FUNCTION_BLOCK "LCB_12x_TablePositioning_V2"   // FB417, SCL
{ S7_Optimized_Access := 'FALSE' }
AUTHOR : Lenze
FAMILY : LCB
NAME : TabPosV2
VERSION : 2.0
   VAR_INPUT
      wHW_IO_Head : Hw_Io;
      i_stcAxisData : "stcLCB_12x_SetAxisData_Sw";
      xEnableInternalControl : Bool;
      iDriveType : Int;
      xDriveEnable : Bool;
      xDriveSetQsp : Bool;
      xResetError : Bool;
      xManualPos : Bool;
      xManualNeg : Bool;
      xHomingSet : Bool;
      xHomingStart : Bool;
      xHomingReset : Bool;
      xProfileStart : Bool;
      xProfileRestart : Bool;
      xProfileReset : Bool;
      xProfilePosStop : Bool;
      wProfileNumberSet : Word := W#16#1;
      xEnableSpeedOverride : Bool;
      rSpeedOverrideSet : Real := 1.0e+2;
      xEnablePositionTeach : Bool;
      rPositionSet : Real;
      xFreeCtrl_1 : Bool;
      xFreeCtrl_2 : Bool;
      xFreeCtrl_3 : Bool;
      xFreeCtrl_4 : Bool;
      xFreeCtrl_5 : Bool;
      xFreeCtrl_6 : Bool;
      xFreeCtrl_7 : Bool;
      xFreeCtrl_8 : Bool;
      wFreeCtrl_1 : Word;
   END_VAR
   VAR_OUTPUT
      xInternalControlActive : Bool;
      xError : Bool;
      xCommunicationOK : Bool;
      xDriveError : Bool;
      xDriveWarning : Bool;
      xDriveReady : Bool;
      xDriveEnabled : Bool;
      xDriveQspActive : Bool;
      xSpeedEqZero : Bool;
      xHomingActive : Bool;
      xHomingDone : Bool;
      xHomePosAvailable : Bool;
      xHomingSensorActivated : Bool;
      xManualActive : Bool;
      xProfileActive : Bool;
      xProfileDone : Bool;
      xProfileInTarget : Bool;
      xHW_LimitSwitchPos : Bool;
      xHW_LimitSwitchNeg : Bool;
      rSpeedActual : Real;
      rPosActual : Real;
      iReadError : Int;
      iWriteError : Int;
      xProfileIsStarting : Bool;   // Drive Application input xPosExecuteIsActive _xFreeState_1 ABS 7/2/2019
      xDirectionSpeedIsCcw : Bool;   // Drive is running anti-clockwise = reverse
      xDriveSafeTorqueOff : Bool;   // Drive Devicestate = SafeTorqueOff
      xFreeState_4 : Bool;
      xFreeState_5 : Bool;
      xFreeState_6 : Bool;
      xFreeState_7 : Bool;
      xFreeState_8 : Bool;
      wFreeState_1 : Word;
      xApplicationError : Bool;   // Table positioning application error, push reset
      xEnabledIsPositionTeach : Bool;   // bPosSetProfilePositionInside the drive
   END_VAR
   VAR
      wFirstPeripherieADR : Word;
      wProfileNumberSetIntern : Word;
      diActPos_p : DInt;
      rAccOverride : Real;
      xDriveEnable_IC : Bool;
      xDriveSetQsp_IC : Bool;
      xResetError_IC : Bool;
      xManualPos_IC : Bool;
      xManualNeg_IC : Bool;
      xHomingSet_IC : Bool;
      xHomingStart_IC : Bool;
      xHomingReset_IC : Bool;
      xProfileStart_IC : Bool;
      xProfileRestart_IC : Bool;
      xProfileReset_IC : Bool;
      xProfilePosStop_IC : Bool;
      xFreeCtrl_1_IC : Bool;
      xFreeCtrl_2_IC : Bool;
      xFreeCtrl_3_IC : Bool;
      xFreeCtrl_4_IC : Bool;
      xFreeCtrl_5_IC : Bool;
      xFreeCtrl_6_IC : Bool;
      xFreeCtrl_7_IC : Bool;
      xFreeCtrl_8_IC : Bool;
      wFreeCtrl_1_IC : Word;
      wProfileNumberSet_IC : Word := W#16#1;
      xwInput AT wProfileNumberSet_IC : Array[0..15] of Bool;
      xEnableSpeedOverride_IC : Bool;
      rSpeedOverrideSet_IC : Real := 1.0e+2;
      xEnablePositionTeach_IC : Bool;
      rPositionSet_IC : Real;
      wOUT : Word;
      xwOut AT wOUT : Array[0..15] of Bool;
      scInternalCtrl84 : Struct
         b8 : Bool;
         b9 : Bool;
         b10 : Bool;
         b11 : Bool;
         b12 : Bool;
         b13 : Bool;
         b14 : Bool;
         b15 : Bool;
         b0 : Bool;
         b1 : Bool;
         b2 : Bool;
         b3 : Bool;
         b4 : Bool;
         b5 : Bool;
         b6 : Bool;
         b7 : Bool;
         awInt : Array[2..6] of Word;
      END_STRUCT;
      scInternalState84 : Struct
         b8 : Bool;
         b9 : Bool;
         b10 : Bool;
         b11 : Bool;
         b12 : Bool;
         b13 : Bool;
         b14 : Bool;
         b15 : Bool;
         b0 : Bool;
         b1 : Bool;
         b2 : Bool;
         b3 : Bool;
         b4 : Bool;
         b5 : Bool;
         b6 : Bool;
         b7 : Bool;
         awInt : Array[2..6] of Word;
      END_STRUCT;
      scInternalCtrl94 : Struct
         b8 : Bool;
         b9 : Bool;
         b10 : Bool;
         b11 : Bool;
         b12 : Bool;
         b13 : Bool;
         b14 : Bool;
         b15 : Bool;
         b0 : Bool;
         b1 : Bool;
         b2 : Bool;
         b3 : Bool;
         b4 : Bool;
         b5 : Bool;
         b6 : Bool;
         b7 : Bool;
         awInt : Array[2..7] of Word;
      END_STRUCT;
      scInternalState94 : Struct
         b8 : Bool;
         b9 : Bool;
         b10 : Bool;
         b11 : Bool;
         b12 : Bool;
         b13 : Bool;
         b14 : Bool;
         b15 : Bool;
         b0 : Bool;
         b1 : Bool;
         b2 : Bool;
         b3 : Bool;
         b4 : Bool;
         b5 : Bool;
         b6 : Bool;
         b7 : Bool;
         awInt : Array[2..7] of Word;
      END_STRUCT;
      dwTemp : DWord;
      rTemp : Real;
      diSetPos : DInt;
   END_VAR
   VAR_TEMP
      Temp_1 : GEOADDR;
      RET : Int;
      tHW_IO : Hw_Any;
   END_VAR
BEGIN
   //#wFirstPeripherieADR:= INT_TO_WORD(#wHW_IO_Head);             
   #iReadError:=0;
   #iWriteError:=0;

   IF #xEnableInternalControl THEN                                    // Interne Steuerung des Reglers
       #xInternalControlActive:=True;
   ELSE                                                               // Steuerung des Reglers über Eingangsvariablen des Bausteins
       #xInternalControlActive:=False;
   END_IF;

   // Keine Interne Steuerung aktiv?
   IF NOT #xEnableInternalControl THEN
       // Eingangssignale auf interne Variablen kopieren
       #xDriveEnable_IC             := #xDriveEnable;
       #xDriveSetQsp_IC             := #xDriveSetQsp;
       #xResetError_IC              := #xResetError;
       #xManualPos_IC               := #xManualPos;
       #xManualNeg_IC               := #xManualNeg;
       #xHomingSet_IC               := #xHomingSet;
       #xHomingStart_IC             := #xHomingStart;
       #xHomingReset_IC             := #xHomingReset;
       #xProfileStart_IC            := #xProfileStart;
       #xProfileRestart_IC          := #xProfileRestart;
       #xProfileReset_IC            := #xProfileReset;
       #xProfilePosStop_IC          := #xProfilePosStop;
       #wProfileNumberSet_IC        := #wProfileNumberSet;
       #xEnableSpeedOverride_IC     := #xEnableSpeedOverride;
       #rSpeedOverrideSet_IC        := #rSpeedOverrideSet;
       #xEnablePositionTeach_IC     := #xEnablePositionTeach;
       #rPositionSet_IC             := #rPositionSet;
       #xFreeCtrl_1_IC              := #xFreeCtrl_1;
       #xFreeCtrl_2_IC              := #xFreeCtrl_2;
       #xFreeCtrl_3_IC              := #xFreeCtrl_3;
       #xFreeCtrl_4_IC              := #xFreeCtrl_4;
       #xFreeCtrl_5_IC              := #xFreeCtrl_5;
       #xFreeCtrl_6_IC              := #xFreeCtrl_6;
       #xFreeCtrl_7_IC              := #xFreeCtrl_7;
       #xFreeCtrl_8_IC              := #xFreeCtrl_8;
       #wFreeCtrl_1_IC              := #wFreeCtrl_1;
   END_IF;

   // HW-Kennung des IO-Moduls für 84/94 ermitteln

   #RET := LOG2GEO(LADDR := #wHW_IO_Head, GEOADDR := #Temp_1); // Aus HW-Kennung des Kopfmoduls den Steckplatz ermitteln
   #Temp_1.SLOT := #Temp_1.SLOT + 1;                           // Slotzähler erhöhen
   #RET := GEO2LOG(GEOADDR := #Temp_1, LADDR => #tHW_IO);      // Aus der Slotnummer die HW_Kennung des ersten Steckplatzes fü

   CASE #iDriveType OF

           // L-Force 8400 Highline / Topline / 8400 Protec Highline
           // Eingangsdaten vom Regler lesen
       2:
           #iReadError := DPRD_DAT(
                                   LADDR := #tHW_IO,
                                   RECORD => #scInternalState84);

           // Statusdaten zuweisen
           #xDriveError := #scInternalState84.b0;
           #xApplicationError := #scInternalState84.b1;
           #xEnabledIsPositionTeach := #scInternalState84.b2;
           #xDriveEnabled := NOT #scInternalState84.b3;
           #xDriveReady := #scInternalState84.b4;
           #xHomingSensorActivated := #scInternalState84.b5;
           #xHomingDone := #scInternalState84.b6;
           #xProfileDone := #scInternalState84.b7;
           #xProfileInTarget := #scInternalState84.b8;
           #xProfileActive := #scInternalState84.b9;
           #xHomePosAvailable := #scInternalState84.b10;
           #xSpeedEqZero := #scInternalState84.b11;
           #xHW_LimitSwitchNeg := #scInternalState84.b12;
           #xHW_LimitSwitchPos := #scInternalState84.b13;
           #xDriveQspActive := #scInternalState84.b14;
           #xDriveWarning := #scInternalState84.b15;

           #xHomingActive := #xHomingStart_IC AND #scInternalState84.b9;

           #rSpeedActual := LIMIT(MN := -199.99, IN := (INT_TO_REAL(WORD_TO_INT(#scInternalState84.awInt[5])) / 163.848), MX := 199.99);
           #diActPos_p := WORD_TO_DINT(#scInternalState84.awInt[3]) + DWORD_TO_DINT(SHL(IN := WORD_TO_DWORD(#scInternalState84.awInt[4]), N := 16));
           // ABS ;-)  #dwTemp := #AxisData.%DBD72;   // AxisData.rPosToUnits
           // ABS done :-) #rTemp := DWORD_TO_REAL(#dwTemp);
           #rPosActual := DINT_TO_REAL(#diActPos_p) * #i_stcAxisData.rPosToUnits;//#rTemp;

           #xProfileIsStarting := WORD_TO_INT((SHR(IN := #scInternalState84.awInt[2], N := 0) AND 16#0001)) > 0;
           #xDirectionSpeedIsCcw := WORD_TO_INT((SHR(IN := #scInternalState84.awInt[2], N := 1) AND 16#0001)) > 0;
           #xDriveSafeTorqueOff := #scInternalState84.awInt[6] >= 16#A00 AND #scInternalState84.awInt[6] <= 16#AFF; //Update TEF 20190917 Devicestate = SafeTorqueOff -> Binary xxxx 1010 xxxx xxxx
           #xFreeState_4 := WORD_TO_INT((SHR(IN := #scInternalState84.awInt[2], N := 3) AND 16#0001)) > 0;
           #xFreeState_5 := WORD_TO_INT((SHR(IN := #scInternalState84.awInt[2], N := 4) AND 16#0001)) > 0;
           #xFreeState_6 := WORD_TO_INT((SHR(IN := #scInternalState84.awInt[2], N := 5) AND 16#0001)) > 0;
           #xFreeState_7 := WORD_TO_INT((SHR(IN := #scInternalState84.awInt[2], N := 6) AND 16#0001)) > 0;
           #xFreeState_8 := WORD_TO_INT((SHR(IN := #scInternalState84.awInt[2], N := 7) AND 16#0001)) > 0;
           #wFreeState_1 := #scInternalState84.awInt[6];

           IF #xHomingStart_IC // Homing ?
               AND NOT #xProfileStart_IC
               AND NOT #xProfileRestart_IC
               AND NOT #xManualPos_IC
               AND NOT #xManualNeg_IC THEN
               // Auswahl 1. Profil für Referenzieren
               #wProfileNumberSet_IC := 1;
               #xManualActive := False;
           ELSIF ((#xManualPos_IC) OR (#xManualNeg_IC)) // Manual ?
               AND NOT #xProfileStart_IC
               AND NOT #xProfileRestart_IC
               AND NOT #xHomingStart_IC
               AND NOT #xHomingSet_IC THEN
               // Auswahl 0. Profil für Handfahren
               #wProfileNumberSet_IC := 0;
               #xManualActive := True;
           ELSE
               #xManualActive := False;

           END_IF;

           IF (NOT #xDriveEnable_IC) OR #xDriveError THEN
               // Merker für Positionieren zurücksetzen
               #xProfileStart_IC := FALSE;
               #xProfileRestart_IC := FALSE;
               #xProfileStart_IC := FALSE;
               #xProfileActive := FALSE;
               #xHomingStart_IC := False;
               #xHomingSet_IC := FALSE;
               #xManualPos_IC := FALSE;
               #xManualPos_IC := FALSE;
               // wProfileNumberSet_IC := 0;        Entfallen mit V1.1    
           END_IF;

           // Steuerdaten zuweisen
           #scInternalCtrl84.b0 := #xProfilePosStop_IC;
           #scInternalCtrl84.b1 := #xProfileRestart_IC AND NOT #xProfilePosStop_IC;
           #scInternalCtrl84.b2 := #xEnablePositionTeach_IC; //update ABS 6/2/2019 AND #xProfileStart_IC;
           #scInternalCtrl84.b3 := NOT #xDriveEnable_IC;
           #scInternalCtrl84.b4 := #xwInput[8];
           #scInternalCtrl84.b5 := #xwInput[9];
           #scInternalCtrl84.b6 := #xwInput[10];
           #scInternalCtrl84.b7 := #xwInput[11];
           #scInternalCtrl84.b8 := #xProfileStart_IC OR #xHomingStart_IC AND NOT #xProfilePosStop_IC;
           #scInternalCtrl84.b9 := #xEnableSpeedOverride_IC;
           #scInternalCtrl84.b10 := #xHomingSet_IC;
           #scInternalCtrl84.b11 := #xResetError_IC;
           #scInternalCtrl84.b12 := #xManualNeg_IC;
           #scInternalCtrl84.b13 := #xManualPos_IC;
           #scInternalCtrl84.b14 := #xHomingReset_IC;
           #scInternalCtrl84.b15 := #xDriveSetQsp_IC;

           // zuweisen der freien Controlbits
           #wOUT := 0;  // Initialisierung
           #xwOut[8] := #xFreeCtrl_1_IC;
           #xwOut[9] := #xFreeCtrl_2_IC;
           #xwOut[10] := #xFreeCtrl_3_IC;
           #xwOut[11] := #xFreeCtrl_4_IC;
           #xwOut[12] := #xFreeCtrl_5_IC;
           #xwOut[13] := #xFreeCtrl_6_IC;
           #xwOut[14] := #xFreeCtrl_7_IC;
           #xwOut[15] := #xFreeCtrl_8_IC;
           #scInternalCtrl84.awInt[2] := #wOUT;

           // limit rSpeedOverride
           #rSpeedOverrideSet_IC := LIMIT(MN := 0.0, IN := #rSpeedOverrideSet_IC, MX := 199.0);
           // scale and Write rSpeedOverride to drive
           IF #xEnableSpeedOverride_IC THEN
               #scInternalCtrl84.awInt[5] := INT_TO_WORD(REAL_TO_INT(#rSpeedOverrideSet_IC * 163.84));
           ELSE
               #scInternalCtrl84.awInt[5] := 16384;
           END_IF;
           //    convert units to increments    
          (* #dwTemp := 1; //#AxisData.%DBD68; // DB SetAxisData.rUnitsToPos
           #rTemp               :=DWORD_TO_REAL(#dwTemp);
          *)

           #diSetPos := REAL_TO_DINT(#rPositionSet_IC * #i_stcAxisData.rUnitsToPos);

           // write to drive*)
           #scInternalCtrl84.awInt[3] := DINT_TO_WORD(#diSetPos);
           #scInternalCtrl84.awInt[4] := DWORD_TO_WORD(SHR(IN := DINT_TO_DWORD(#diSetPos), N := 16));
           #scInternalCtrl84.awInt[6] := #wFreeCtrl_1_IC;

           // Ausgangsdaten zum Regler schreiben                         
           #iWriteError := DPWR_DAT(
                                    LADDR := #tHW_IO,
                                    RECORD := #scInternalCtrl84);

           #xError := (#iReadError <> 0) OR (#iWriteError <> 0)
           OR NOT ((#iDriveType <> 2) OR (#iDriveType <> 11))
           OR (WORD_TO_INT(#wProfileNumberSet_IC) > 15)
           OR (WORD_TO_INT(#wProfileNumberSet_IC) < 0);




           // L-Force 9400 Highline 
           // Eingangsdaten vom Regler lesen
       11:
           #iReadError := DPRD_DAT(
                                   LADDR := #tHW_IO,
                                   RECORD => #scInternalState94);

           // Statusdaten zuweisen
           #xDriveError := #scInternalState94.b0;
           #xDriveEnabled := NOT #scInternalState94.b1;
           #xDriveReady := #scInternalState94.b2;
           #xDriveQspActive := #scInternalState94.b3;
           #xSpeedEqZero := #scInternalState94.b4;
           #xHomingActive := #scInternalState94.b5;
           #xHomingDone := #scInternalState94.b6;
           #xHomePosAvailable := #scInternalState94.b7;
           #xManualActive := #scInternalState94.b8;
           #xDriveWarning := #scInternalState94.b9;
           #xProfileActive := #scInternalState94.b10;
           #xProfileDone := #scInternalState94.b11;
           #xProfileInTarget := #scInternalState94.b12;
           // xHomeSwitch      :=scInternalState94.b13;
           #xHW_LimitSwitchPos := #scInternalState94.b14;
           #xHW_LimitSwitchNeg := #scInternalState94.b15;

           #rSpeedActual := LIMIT(MN := -199.99, IN := (INT_TO_REAL(WORD_TO_INT(#scInternalState94.awInt[2])) / 163.848), MX := 199.99);
           #diActPos_p := WORD_TO_DINT(#scInternalState94.awInt[4]) + DWORD_TO_DINT(SHL(IN := WORD_TO_DWORD(#scInternalState94.awInt[3]), N := 16));
           // ABS;-) #dwTemp := #AxisData.%DBD72;   // AxisData.rPosToUnits
           // ABS :-) #rTemp := DWORD_TO_REAL(#dwTemp);
           #rPosActual := DINT_TO_REAL(#diActPos_p) * #i_stcAxisData.rPosToUnits;//#rTemp;

           #xProfileIsStarting := WORD_TO_INT((SHR(IN := #scInternalState94.awInt[6], N := 0) AND 16#0001)) > 0;
           #xDirectionSpeedIsCcw := WORD_TO_INT((SHR(IN := #scInternalState94.awInt[6], N := 1) AND 16#0001)) > 0;
           #xDriveSafeTorqueOff := WORD_TO_INT((SHR(IN := #scInternalState94.awInt[6], N := 2) AND 16#0001)) > 0;
           #xFreeState_4 := WORD_TO_INT((SHR(IN := #scInternalState94.awInt[6], N := 3) AND 16#0001)) > 0;
           #xFreeState_5 := WORD_TO_INT((SHR(IN := #scInternalState94.awInt[6], N := 4) AND 16#0001)) > 0;
           #xFreeState_6 := WORD_TO_INT((SHR(IN := #scInternalState94.awInt[6], N := 5) AND 16#0001)) > 0;
           #xFreeState_7 := WORD_TO_INT((SHR(IN := #scInternalState94.awInt[6], N := 6) AND 16#0001)) > 0;
           #xFreeState_8 := WORD_TO_INT((SHR(IN := #scInternalState94.awInt[6], N := 7) AND 16#0001)) > 0;
           #wFreeState_1 := #scInternalState94.awInt[5];

           IF (NOT #xDriveEnable_IC) OR #xDriveError THEN
               // Merker für Positionieren zurücksetzen
               #xProfileStart_IC := FALSE;
               #xProfileRestart_IC := FALSE;
               #xProfileStart_IC := FALSE;
               #xProfileActive := FALSE;
               #xHomingStart_IC := False;
               #xHomingSet_IC := FALSE;
               #xManualPos_IC := FALSE;
               #xManualPos_IC := FALSE;
               // wProfileNumberSet_IC := 1;    entfallen mit V1.1        
           END_IF;

           // Steuerdaten zuweisen
           #scInternalCtrl94.b0 := NOT #xDriveEnable_IC;
           #scInternalCtrl94.b1 := #xDriveSetQsp_IC;
           #scInternalCtrl94.b2 := #xEnablePositionTeach_IC;
           #scInternalCtrl94.b3 := #xHomingStart_IC;
           #scInternalCtrl94.b4 := #xHomingReset_IC;
           #scInternalCtrl94.b5 := #xProfileActive OR #xProfileStart_IC;
           #scInternalCtrl94.b6 := #xProfileStart_IC AND NOT #xProfilePosStop_IC;
           #scInternalCtrl94.b7 := #xProfileRestart_IC AND NOT #xProfilePosStop_IC;
           #scInternalCtrl94.b8 := #xProfileReset_IC;
           #scInternalCtrl94.b9 := #xEnableSpeedOverride_IC;
           #scInternalCtrl94.b10 := #xResetError_IC;
           #scInternalCtrl94.b11 := False; // Spare Set Error
           #scInternalCtrl94.b12 := #xHomingSet_IC;
           #scInternalCtrl94.b13 := False; // Spare
           #scInternalCtrl94.b14 := #xManualPos_IC;
           #scInternalCtrl94.b15 := #xManualNeg_IC;

           // zuweisen der freien Controlbits
           #wOUT := 0;  // Initialisierung
           #xwOut[8] := #xFreeCtrl_1_IC;
           #xwOut[9] := #xFreeCtrl_2_IC;
           #xwOut[10] := #xFreeCtrl_3_IC;
           #xwOut[11] := #xFreeCtrl_4_IC;
           #xwOut[12] := #xFreeCtrl_5_IC;
           #xwOut[13] := #xFreeCtrl_6_IC;
           #xwOut[14] := #xFreeCtrl_7_IC;
           #xwOut[15] := #xFreeCtrl_8_IC;
           #scInternalCtrl94.awInt[6] := #wOUT;
           #scInternalCtrl94.awInt[7] := #wFreeCtrl_1_IC;

           // limit rSpeedOverride
           #rSpeedOverrideSet_IC := LIMIT(MN := 0.0, IN := #rSpeedOverrideSet_IC, MX := 199.0);
           // scale and Write rSpeedOverride to drive
           IF #xEnableSpeedOverride_IC THEN
               #scInternalCtrl94.awInt[2] := INT_TO_WORD(REAL_TO_INT(#rSpeedOverrideSet_IC * 163.84));
           ELSE
               #scInternalCtrl94.awInt[2] := 16384;
           END_IF;
           // convert units to increments    
           //ABS :-)  #dwTemp := #AxisData.%DBD68; // DB SetAxisData.rUnitsToPos
           //ABS :-)  #rTemp := DWORD_TO_REAL(#dwTemp);
           #diSetPos := REAL_TO_DINT(#rPositionSet_IC * #i_stcAxisData.rUnitsToPos);//#rTemp);

           // write to drive*)
           #scInternalCtrl94.awInt[4] := DINT_TO_WORD(#diSetPos);
           #scInternalCtrl94.awInt[3] := DWORD_TO_WORD(SHR(IN := DINT_TO_DWORD(#diSetPos), N := 16));

           // limit  ProfileNumber and write To Drive      
           #scInternalCtrl94.awInt[5] := INT_TO_WORD(LIMIT(MN := 1, IN := WORD_TO_INT(#wProfileNumberSet_IC), MX := 75));

           // Ausgangsdaten zum Regler schreiben                         
           #iWriteError := DPWR_DAT(
                                    LADDR := #tHW_IO,
                                    RECORD := #scInternalCtrl94);

           #xError := (#iReadError <> 0) OR (#iWriteError <> 0)
           OR NOT ((#iDriveType <> 1) OR (#iDriveType <> 2) OR (#iDriveType <> 11))
           OR (WORD_TO_INT(#wProfileNumberSet_IC) > 75)
           OR (WORD_TO_INT(#wProfileNumberSet_IC) < 1);

       ELSE:
           #xError := True;
   END_CASE;

   IF (#iReadError <> 0) OR (#iWriteError <> 0) THEN
       #xCommunicationOK:=false;
   ELSE
       #xCommunicationOK:=True;
   END_IF;
END_FUNCTION_BLOCK

FUNCTION_BLOCK "LCB_12x_SetAxisData"   // FB443, SCL
{ S7_Optimized_Access := 'FALSE' }
AUTHOR : Lenze
FAMILY : LCB
NAME : SetAxisD
VERSION : 1.0
   VAR_INPUT
      rFeedConstant : Real := 3.6e+2;
      rCycleLength : Real := 3.6e+2;
      diGearNumerator : DInt := L#1;
      diGearDenominator : DInt := L#1;
      rReferenceSpeed : Real := 1.8e+5;
      rReferenceTorque : Real := 1.0e+0;
      sAxisName : String[16] := 'MyAxis';
      rResolution : Real := 16.0;
   END_VAR
   VAR_OUTPUT
      AxisData : "stcLCB_12x_SetAxisData_Sw";
   END_VAR
   VAR_IN_OUT
      xModeUnlimited : Bool := TRUE;
      xModeLimited : Bool;
      xModeModulo : Bool;
   END_VAR
   VAR
      rInvFeedConstant : Real;
      diReferenceSpeed_s : DInt;
      rEncoderGear : Real;
      rInvEncoderGear : Real;
      diCycleLength_p : DInt;
      rUnitsToPos : Real;
      rPosToUnits : Real;
      rUnitsToSpeed : Real;
      rSpeedToUnits : Real;
      rTimeUnit : Real := 6.0e+1;
      rFeedConstantOld : Real;
      rCycleLengthOld : Real;
      diGearNumeratorOld : DInt := L#2;
      diGearDenominatorOld : DInt := L#2;
      rReferenceSpeedOld : Real;
      rResolutionOld : Real := 1.0;
      xModeUnlimitedOld : Bool;
      xModeLimitedOld : Bool;
      xModeModuloOld : Bool;
   END_VAR
BEGIN

       IF #xModeUnlimited= True THEN #xModeLimited:= False; #xModeModulo:= False;
           ELSIF #xModeLimited= True THEN #xModeUnlimited:= False; #xModeModulo:= False;
               ELSIF #xModeModulo= True THEN #xModeUnlimited:= False; #xModeLimited:= False;
       END_IF; 
       IF ((#rFeedConstantOld <> #rFeedConstant) OR
           (#diGearNumeratorOld <> #diGearNumerator) OR
           (#diGearDenominatorOld <> #diGearDenominator) OR
           (#rCycleLengthOld <> #rCycleLength) OR
           (#xModeUnlimitedOld <> #xModeUnlimited) OR
           (#xModeLimitedOld <> #xModeLimited) OR
           (#xModeModuloOld <> #xModeModulo) OR
           (#rResolutionOld <> #rResolution) OR
           (#rReferenceSpeedOld <> #rReferenceSpeed)) THEN


           #rInvFeedConstant := 1.0 / #rFeedConstant;

       (* Achsdatenberechnung starten *)
       (* Getriebefaktor *)
           #rEncoderGear:=DINT_TO_REAL(#diGearNumerator) / DINT_TO_REAL(#diGearDenominator);
           #rInvEncoderGear:= 1.0 / #rEncoderGear;
       (* Umrechenfaktor Units -> _p bestimmen *)
           #rUnitsToPos := (#rInvFeedConstant * #rEncoderGear) * (2**#rResolution);
       (* Umrechenfaktor _p -> Units bestimmen *)
           #rPosToUnits := 1.0 / #rUnitsToPos;
       (* Umrechenfaktor Units->_s bestimmen *)
           #rUnitsToSpeed := #rInvFeedConstant * #rEncoderGear;
     //  (* mal 2^32 (eine Umdrehung) *)
     //      rUnitsToSpeed := rUnitsToSpeed * 2**32;
       (* durch Zeiteinheit teilen *)
           #rUnitsToSpeed := #rUnitsToSpeed * #rTimeUnit;
       (* Umrechenfaktor _s -> Units bestimmen *)
           #rSpeedToUnits := 1.0 / #rUnitsToSpeed;
       (*Referenzgeschwindigkeit bestimmen *)
           #diReferenceSpeed_s := REAL_TO_DINT(#rReferenceSpeed * #rUnitsToSpeed);

           IF #xModeModulo THEN
               #diCycleLength_p := REAL_TO_DINT(#rCycleLength * #rUnitsToPos) ;
           ELSE
               #diCycleLength_p := 0;
           END_IF;

       // sichern der aktuellen Werte für Änderungsvergleich
           #rFeedConstantOld     :=#rFeedConstant     ;
           #rCycleLengthOld      :=#rCycleLength      ;    
           #diGearNumeratorOld   :=#diGearNumerator   ;
           #diGearDenominatorOld :=#diGearDenominator ;
           #rReferenceSpeedOld   :=#rReferenceSpeed   ;
           #xModeUnlimitedOld    :=#xModeUnlimited    ;
           #xModeLimitedOld      :=#xModeLimited      ;
           #xModeModuloOld       :=#xModeModulo       ;
           #rResolutionOld      :=#rResolution      ;  

       END_IF;

   //Write to global output status
       #AxisData.rUnitsToPos := #rUnitsToPos;
       #AxisData.rPosToUnits := #rPosToUnits;
END_FUNCTION_BLOCK

(* ===== HMI "HMI_RT_1" =====
system functions are stored by id; their names below are inferred from use
connection "HMI_Connection_1": ETHERNET, S7_1200_OMS

HMI tags "Default tag table"
   "VIS_CmDrvSerPos_stc_Indicators_Status_IsEnabled" : Bool = PLC VIS_CmDrvSerPos.stc.Indicators.Status.IsEnabled, 1 s
   "VIS_CmDrvSerPos_stc_Commands_Enable" : Bool = PLC VIS_CmDrvSerPos.stc.Commands.Enable, 1 s
   "VIS_CmDrvSerPos_stc_Commands_JogFwdCwUpLoading" : Bool = PLC VIS_CmDrvSerPos.stc.Commands.JogFwdCwUpLoading, 1 s
   "VIS_CmDrvSerPos_stc_Commands_JogRevCcwDownUnloading" : Bool = PLC VIS_CmDrvSerPos.stc.Commands.JogRevCcwDownUnloading, 1 s
   "VIS_CmDrvSerPos_stc_Indicators_Status_BusyJogFwdCwUpLoading" : Bool = PLC VIS_CmDrvSerPos.stc.Indicators.Status.BusyJogFwdCwUpLoading, 1 s
   "VIS_CmDrvSerPos_stc_Indicators_Status_BusyJogRevCcwDownUnloading" : Bool = PLC VIS_CmDrvSerPos.stc.Indicators.Status.BusyJogRevCcwDownUnloading, 1 s
   "VIS_CmDrvSerPos_stc_Commands_PbReset" : Bool = PLC VIS_CmDrvSerPos.stc.Commands.PbReset, 1 s
   "VIS_CmDrvSerPos_stc_Indicators_PushButtons_PbReset" : Bool = PLC VIS_CmDrvSerPos.stc.Indicators.PushButtons.PbReset, 1 s
   "VIS_CmDrvSerPos_stc_Commands_StartHoming" : Bool = PLC VIS_CmDrvSerPos.stc.Commands.StartHoming, 1 s
   "VIS_CmDrvSerPos_stc_Indicators_Status_IsHomed" : Bool = PLC VIS_CmDrvSerPos.stc.Indicators.Status.IsHomed, 1 s
   "VIS_CmDrvSerPos_stc_Commands_StartExecuteAutomatic" : Bool = PLC VIS_CmDrvSerPos.stc.Commands.StartExecuteAutomatic, 1 s
   "VIS_CmDrvSerPos_stc_Commands_StopHoming" : Bool = PLC VIS_CmDrvSerPos.stc.Commands.StopHoming, 1 s
   "VIS_CmDrvSerPos_stc_Recipe_rSpPosition_Units" : Real = PLC VIS_CmDrvSerPos.stc.Recipe.rSpPosition_Units, 1 s
   "VIS_CmDrvSerPos_stc_SD_ProcessValue_rPvPosition_Units" : Real = PLC VIS_CmDrvSerPos.stc.SD.ProcessValue.rPvPosition_Units, 1 s
   "VIS_CmDrvSerPos_stc_Indicators_PushButtons_StopHoming" : Bool = PLC VIS_CmDrvSerPos.stc.Indicators.PushButtons.StopHoming, 1 s
   "VIS_CmDrvSerPos_stc_Indicators_PushButtons_StartHoming" : Bool = PLC VIS_CmDrvSerPos.stc.Indicators.PushButtons.StartHoming, 1 s
   "VIS_CmDrvSerPos_stc_Indicators_PushButtons_StartExecuteAutomatic" : Bool = PLC VIS_CmDrvSerPos.stc.Indicators.PushButtons.StartExecuteAutomatic, 1 s
   "VIS_CmDrvSerPos_stc_Indicators_Status_IsAtTargetPosSpeed" : Bool = PLC VIS_CmDrvSerPos.stc.Indicators.Status.IsAtTargetPosSpeed, 1 s
   "VIS_CmDrvSerPos_stc_Commands_StopExecuteAutomatic" : Bool = PLC VIS_CmDrvSerPos.stc.Commands.StopExecuteAutomatic, 1 s
   "VIS_CmDrvSerPos_stc_Indicators_PushButtons_StopExecuteAutomatic" : Bool = PLC VIS_CmDrvSerPos.stc.Indicators.PushButtons.StopExecuteAutomatic, 1 s
   "VIS_CmDrvSerPos_stc_SD_ErrorWarning_bErrorTripped" : Bool = PLC VIS_CmDrvSerPos.stc.SD.ErrorWarning.bErrorTripped, 1 s
   "VIS_CmDrvSerPos_stc_SD_ErrorWarning_bWarningTripped" : Bool = PLC VIS_CmDrvSerPos.stc.SD.ErrorWarning.bWarningTripped, 1 s
   "VIS_CmDrvSerPos_stc_SD_bRFR" : Bool = PLC VIS_CmDrvSerPos.stc.SD.bRFR, 1 s
   "VIS_CmDrvSerPos_stc_SD_ErrorWarning_wError" : Word = PLC VIS_CmDrvSerPos.stc.SD.ErrorWarning.wError, 1 s
   "VIS_CmDrvSerPos_stc_SD_ErrorWarning_wWarning" : Word = PLC VIS_CmDrvSerPos.stc.SD.ErrorWarning.wWarning, 1 s
   "VIS_CmDrvSerPos_stc_bLimitsSwitchPositiveActivated" : Bool = PLC VIS_CmDrvSerPos.stc.bLimitsSwitchPositiveActivated, 1 s
   "VIS_CmDrvSerPos_stc_bLimitsSwitchNegativeActivated" : Bool = PLC VIS_CmDrvSerPos.stc.bLimitsSwitchNegativeActivated, 1 s
   "VIS_CmDrvSerPos_stc_bHomingSensorActivated" : Bool = PLC VIS_CmDrvSerPos.stc.bHomingSensorActivated, 1 s
   "VIS_CmDrvSerPos_stc_CD_iModeSet" : Int = PLC VIS_CmDrvSerPos.stc.CD.iModeSet, 1 s
   "VIS_CmDrvSerPos_stc_Commands_ModeChange" : Bool = PLC VIS_CmDrvSerPos.stc.Commands.ModeChange, 1 s
   "DB_CmDrvSerPos_CD_iModeSet" : Int = PLC DB_CmDrvSerPos.CD.iModeSet, 1 s
   "DB_CmDrvSerPos_CD_Commands_ModeChange" : Bool = PLC DB_CmDrvSerPos.CD.Commands.ModeChange, 1 s
   "VIS_CmDrvSerPos_stc_SD_iModeActual" : Int = PLC VIS_CmDrvSerPos.stc.SD.iModeActual, 1 s
   "VIS_CmDrvSerPos_stc_Commands_Disable" : Bool = PLC VIS_CmDrvSerPos.stc.Commands.Disable, 1 s
   "VIS_CmDrvSerPos_stc_SD_iModuleState" : Int = PLC VIS_CmDrvSerPos.stc.SD.iModuleState, 1 s
   "VIS_CmDrvSerPos_stc_SD_bExecuting" : Bool = PLC VIS_CmDrvSerPos.stc.SD.bExecuting, 1 s
   "VIS_CmDrvSerPos_stc_Commands_EnableReleaseErrorWarning" : Bool = PLC VIS_CmDrvSerPos.stc.Commands.EnableReleaseErrorWarning, 1 s
   "VIS_CmDrvSerPos_stc_Commands_DisableReleaseErrorWarning" : Bool = PLC VIS_CmDrvSerPos.stc.Commands.DisableReleaseErrorWarning, 1 s
   "VIS_CmDrvSerPos_stc_Commands_ExecuteLoadRecipe" : Bool = PLC VIS_CmDrvSerPos.stc.Commands.ExecuteLoadRecipe, 1 s
   "VIS_CmDrvSerPos_stc_SD_ErrorWarningReleased" : Bool = PLC VIS_CmDrvSerPos.stc.SD.ErrorWarningReleased AT %DB1.DBX0.0, 1 s
   "di_FeedbackEmStop" : Bool = PLC di_FeedbackEmStop AT %I0.4, 1 s
   "VIS_CmDrvSerPos_stc_Indicators_PushButtons_Enable" : Bool = PLC VIS_CmDrvSerPos.stc.Indicators.PushButtons.Enable, 1 s
   "VIS_CmDrvSerPos_stc_Indicators_PushButtons_Disable" : Bool = PLC VIS_CmDrvSerPos.stc.Indicators.PushButtons.Disable, 1 s
   "VIS_CmDrvSerPos_stc_Indicators_PushButtons_ExecuteLoadRecipe" : Bool = PLC VIS_CmDrvSerPos.stc.Indicators.PushButtons.ExecuteLoadRecipe, 1 s
   "VIS_CmDrvSerPos_stc_Settings_rSpLimitH_Units" : Real = PLC VIS_CmDrvSerPos.stc.Settings.rSpLimitH_Units, 1 s
   "VIS_CmDrvSerPos_stc_Settings_rSpLimitL_Units" : Real = PLC VIS_CmDrvSerPos.stc.Settings.rSpLimitL_Units, 1 s
   "VIS_CmDrvSerPos_stc_Settings_rSpPositionOffset_Units" : Real = PLC VIS_CmDrvSerPos.stc.Settings.rSpPositionOffset_Units, 1 s
   "VIS_CmDrvSerPos_stc_Settings_iSetUnits" : Int = PLC VIS_CmDrvSerPos.stc.Settings.iSetUnits, 1 s

text list "Mode": 0 'Undefined'; 1 'AutoInline'; 2 'AutoStandalone'; 3 'Manual'; 4 'Service'; 5 'SingleStep'

screen "Screen_1" 800x480, template "Template_1"
   Rectangle "Rectangle_1" at 17,147 size 20x90
      Appearance <- "VIS_CmDrvSerPos_stc_Indicators_PushButtons_Enable"
   Button "Button_1" at 34,147 size 150x90; TextOff 'Enable'
      on Release: ResetBit("VIS_CmDrvSerPos_stc_Commands_Enable")
      on Press: SetBit("VIS_CmDrvSerPos_stc_Commands_Enable")
   Rectangle "Rectangle_2" at 196,376 size 20x90
      Appearance <- "VIS_CmDrvSerPos_stc_Indicators_Status_BusyJogFwdCwUpLoading"
   Button "Button_2" at 213,376 size 150x90; TextOff 'Fwd/Up'
      on Release: ResetBit("VIS_CmDrvSerPos_stc_Commands_JogFwdCwUpLoading")
      on Press: SetBit("VIS_CmDrvSerPos_stc_Commands_JogFwdCwUpLoading")
   Rectangle "Rectangle_3" at 14,376 size 20x90
      Appearance <- "VIS_CmDrvSerPos_stc_Indicators_Status_BusyJogRevCcwDownUnloading"
   Button "Button_3" at 31,376 size 150x90; TextOff 'Rev/Down'
      on Release: ResetBit("VIS_CmDrvSerPos_stc_Commands_JogRevCcwDownUnloading")
      on Press: SetBit("VIS_CmDrvSerPos_stc_Commands_JogRevCcwDownUnloading")
   Rectangle "Rectangle_4" at 17,246 size 20x90
      Appearance <- "VIS_CmDrvSerPos_stc_Indicators_PushButtons_PbReset"
   Button "Button_4" at 34,246 size 150x90; TextOff 'Reset'
      on Release: ResetBit("VIS_CmDrvSerPos_stc_Commands_PbReset")
      on Press: SetBit("VIS_CmDrvSerPos_stc_Commands_PbReset")
   Button "Button_5" at 213,246 size 150x90; TextOff 'QuickStop'
   Rectangle "Rectangle_6" at 389,376 size 20x90
      Appearance <- "VIS_CmDrvSerPos_stc_Indicators_PushButtons_StartHoming"
   Button "Button_6" at 406,376 size 150x90; TextOff 'Start'
      on Release: ResetBit("VIS_CmDrvSerPos_stc_Commands_StartHoming")
      on Press: SetBit("VIS_CmDrvSerPos_stc_Commands_StartHoming")
   Rectangle "Rectangle_7" at 390,150 size 20x90
      Appearance <- "VIS_CmDrvSerPos_stc_Indicators_PushButtons_StartExecuteAutomatic"
   Button "Button_7" at 407,150 size 150x90; TextOff 'Enable'
      on Release: ResetBit("VIS_CmDrvSerPos_stc_Commands_StartExecuteAutomatic")
      on Press: SetBit("VIS_CmDrvSerPos_stc_Commands_StartExecuteAutomatic")
   TextField "Text field_1" at 525,349 size 73x23; Text 'Homing'
   TextField "Text field_2" at 169,349 size 36x23; Text 'Jog'
   Button "Button_8" at 569,376 size 150x90; TextOff 'Stop'
      on Release: ResetBit("VIS_CmDrvSerPos_stc_Commands_StopHoming")
      on Press: SetBit("VIS_CmDrvSerPos_stc_Commands_StopHoming")
   TextField "Text field_3" at 471,121 size 152x23; Text 'Position Control'
   IOField "I/O field_1" at 414,248 size 141x39; FormatPattern s999.9; Unit mm
      ProcessValue <- "VIS_CmDrvSerPos_stc_Recipe_rSpPosition_Units"
   IOField "I/O field_2" at 415,293 size 140x41; FormatPattern s999.9; Unit mm
      ProcessValue <- "VIS_CmDrvSerPos_stc_SD_ProcessValue_rPvPosition_Units"
   Rectangle "Rectangle_12" at 620,350 size 20x24
      Appearance <- "VIS_CmDrvSerPos_stc_Indicators_Status_IsHomed"
   Button "Button_9" at 573,150 size 150x90; TextOff 'Disable'
      on Release: ResetBit("VIS_CmDrvSerPos_stc_Commands_StopExecuteAutomatic")
      on Press: SetBit("VIS_CmDrvSerPos_stc_Commands_StopExecuteAutomatic")
   Rectangle "Rectangle_14" at 716,150 size 20x90
      Appearance <- "VIS_CmDrvSerPos_stc_Indicators_PushButtons_StopExecuteAutomatic"
   TextField "Text field_6" at 385,255 size 28x23; Text 'SP'
   TextField "Text field_7" at 385,300 size 29x23; Text 'PV'
   Button "Button_10" at 6,52 size 739x52; TextOff 'Enable'
   TextField "Text field_8" at 315,17 size 143x23; Text 'CmDriveSerPos'
   TextField "Text field_9" at 151,119 size 76x23; Text 'General'
   Rectangle "Rectangle_10" at 716,376 size 20x90
      Appearance <- "VIS_CmDrvSerPos_stc_Indicators_PushButtons_StopHoming"
   Button "Button_11" at 747,417 size 51x56; TextOff 'Enable'; PictureOff "Down_Arrow"
      on Release: ActivateScreen("Screen_2", 0)
   Button "Button_12" at 747,112 size 51x56; TextOff 'Enable'; PictureOff "Up_Arrow"
      on Release: ActivateScreen("Screen_2", 0)
   TextField "Text field_10" at 772,280 size 16x23; Text '3'
   TextField "Text field_11" at 751,280 size 16x23; Text '1'
   Button "Button_13" at 747,52 size 50x52; TextOff 'CmValveCtrl'; PictureOff "Home"
      on Release: ActivateScreen("Main_Screen", 0)
   IOField "I/O field_3" at 18,117 size 44x26; FormatPattern 9999
      ProcessValue <- "VIS_CmDrvSerPos_stc_SD_iModuleState"
   Button "Button_15" at 573,246 size 145x40; TextOff 'Single Step'
      on Release: ResetBit("VIS_CmDrvSerPos_stc_Commands_ExecuteLoadRecipe")
      on Press: SetBit("VIS_CmDrvSerPos_stc_Commands_ExecuteLoadRecipe")
   TextField "Text field_4" at 645,352 size 94x18; Text 'HomingDone'
   Rectangle "Rectangle_16" at 620,122 size 20x24
      Appearance <- "VIS_CmDrvSerPos_stc_Indicators_Status_IsAtTargetPosSpeed"
   TextField "Text field_5" at 645,125 size 66x18; Text 'InTarget'
   Rectangle "Rectangle_13" at 254,119 size 20x24
      Appearance <- "VIS_CmDrvSerPos_stc_Indicators_Status_IsEnabled"
   TextField "Text field_12" at 279,122 size 60x18; Text 'Enabled'
   Rectangle "Rectangle_17" at 196,147 size 20x90
      Appearance <- "VIS_CmDrvSerPos_stc_Indicators_PushButtons_Disable"
   Button "Button_14" at 212,147 size 150x90; TextOff 'Disable'
      on Release: ResetBit("VIS_CmDrvSerPos_stc_Commands_Disable")
      on Press: SetBit("VIS_CmDrvSerPos_stc_Commands_Disable")
   Rectangle "Rectangle_18" at 716,246 size 20x90
      Appearance <- "VIS_CmDrvSerPos_stc_Indicators_PushButtons_ExecuteLoadRecipe"
   Button "Button_16" at 573,296 size 145x40; TextOff 'Automatic'
      on Press: SetBit("VIS_CmDrvSerPos_stc_Commands_ExecuteLoadRecipe")

screen "Screen_2" 800x480, template "Template_1"
   TextField "Text field_3" at 458,119 size 232x23; Text 'Status Sequence Stepper'
   Button "Button_10" at 6,52 size 739x52; TextOff 'Enable'
   TextField "Text field_8" at 315,17 size 143x23; Text 'CmDriveSerPos'
   TextField "Text field_9" at 149,119 size 108x23; Text 'Status OEM'
   Button "Button_12" at 747,417 size 51x56; TextOff 'Enable'; PictureOff "Down_Arrow"
      on Release: ActivateScreen("Screen_3", 0)
   Button "Button_13" at 747,112 size 51x56; TextOff 'Enable'; PictureOff "Up_Arrow"
      on Release: ActivateScreen("Screen_1", 0)
   TextField "Text field_10" at 772,280 size 16x23; Text '3'
   TextField "Text field_11" at 750,280 size 16x23; Text '2'
   Ellipse "Ellipse_1" at 397,149 size 28x28
      Appearance <- "VIS_CmDrvSerPos_stc_Indicators_Status_IsEnabled"
   TextField "Text field_2" at 435,152 size 77x23; Text 'Enabled'
   Ellipse "Ellipse_2" at 24,184 size 28x28
      Appearance <- "VIS_CmDrvSerPos_stc_SD_ErrorWarning_bErrorTripped"
   TextField "Text field_12" at 60,187 size 51x23; Text 'Error'
   Ellipse "Ellipse_3" at 398,189 size 28x28
      Appearance <- "VIS_CmDrvSerPos_stc_Indicators_Status_BusyJogRevCcwDownUnloading"
   TextField "Text field_13" at 436,190 size 125x23; Text 'Jog Fwd busy'
   Ellipse "Ellipse_4" at 397,229 size 28x28
      Appearance <- "VIS_CmDrvSerPos_stc_Indicators_Status_BusyJogRevCcwDownUnloading"
   TextField "Text field_14" at 437,229 size 123x23; Text 'Jog Rev busy'
   Ellipse "Ellipse_5" at 397,267 size 28x28
      Appearance <- "VIS_CmDrvSerPos_stc_SD_iModuleState"
   TextField "Text field_1" at 440,267 size 120x23; Text 'Homing busy'
   Ellipse "Ellipse_6" at 397,303 size 28x28
      Appearance <- "VIS_CmDrvSerPos_stc_SD_iModuleState"
   TextField "Text field_4" at 441,306 size 166x23; Text 'Position Ctrl busy'
   Ellipse "Ellipse_7" at 24,146 size 28x28
      Appearance <- "VIS_CmDrvSerPos_stc_SD_ErrorWarning_bWarningTripped"
   TextField "Text field_5" at 59,149 size 80x23; Text 'Warning'
   Ellipse "Ellipse_8" at 23,261 size 28x28
      Appearance <- "VIS_CmDrvSerPos_stc_SD_bRFR"
   TextField "Text field_6" at 60,264 size 115x23; Text 'Drive Ready'
   Ellipse "Ellipse_9" at 23,222 size 28x28
      Appearance <- "VIS_CmDrvSerPos_stc_Indicators_Status_IsEnabled"
   TextField "Text field_7" at 60,225 size 131x23; Text 'Drive Enabled'
   Ellipse "Ellipse_10" at 23,302 size 28x28
      Appearance <- "VIS_CmDrvSerPos_stc_Indicators_Status_IsHomed"
   TextField "Text field_15" at 61,306 size 67x23; Text 'Homed'
   IOField "I/O field_1" at 162,378 size 80x40; FormatPattern 99999
      ProcessValue <- "VIS_CmDrvSerPos_stc_SD_ErrorWarning_wWarning"
   TextField "Text field_17" at 18,388 size 135x23; Text 'Warning code:'
   IOField "I/O field_2" at 162,425 size 80x40; FormatPattern 99999
      ProcessValue <- "VIS_CmDrvSerPos_stc_SD_ErrorWarning_wError"
   TextField "Text field_16" at 20,431 size 106x23; Text 'Error code:'
   Ellipse "Ellipse_11" at 397,359 size 28x28
      Appearance <- "VIS_CmDrvSerPos_stc_bLimitsSwitchPositiveActivated"
   TextField "Text field_18" at 441,362 size 155x23; Text 'Limit Switch Pos'
   Ellipse "Ellipse_12" at 397,394 size 28x28
      Appearance <- "VIS_CmDrvSerPos_stc_bLimitsSwitchNegativeActivated"
   TextField "Text field_19" at 441,397 size 158x23; Text 'Limit Switch Neg'
   Ellipse "Ellipse_13" at 397,429 size 28x28
      Appearance <- "VIS_CmDrvSerPos_stc_bHomingSensorActivated"
   TextField "Text field_20" at 442,432 size 140x23; Text 'Homing Sensor'
   Button "Button_1" at 747,52 size 50x52; TextOff 'CmValveCtrl'; PictureOff "Home"
      on Release: ActivateScreen("Main_Screen", 0)
   Ellipse "Ellipse_14" at 22,341 size 28x28
      Appearance <- "VIS_CmDrvSerPos_stc_SD_bExecuting"
   TextField "Text field_21" at 60,345 size 94x23; Text 'Executing'
   Button "Button_2" at 176,155 size 81x57; TextOff 'Enable'
      on Release: ResetBit("VIS_CmDrvSerPos_stc_Commands_EnableReleaseErrorWarning")
      on Press: SetBit("VIS_CmDrvSerPos_stc_Commands_EnableReleaseErrorWarning")
   Button "Button_3" at 268,155 size 81x57; TextOff 'Disable'
      on Release: ResetBit("VIS_CmDrvSerPos_stc_Commands_DisableReleaseErrorWarning")
      on Press: SetBit("VIS_CmDrvSerPos_stc_Commands_DisableReleaseErrorWarning")
   Rectangle "Rectangle_13" at 160,154 size 20x58
      Appearance <- "VIS_CmDrvSerPos_stc_SD_ErrorWarningReleased"

Template "Template_1" 800x480
   TextField "Text field_1" at 762,279 size 15x23; Text '/'

screen "HMI_Settings" 800x480
   TextField "Text field_8" at 346,17 size 122x23; Text 'HMI Settings'
   Button "HmiScreenItemData" at 23,131 size 159x47; TextOn 'SIMATIC PLC system diagnos...'; TextOff 'SIMATIC PLC system diagnos...'; PictureOn "Navigates to SIMATIC PLC system diagnostics for TP700 Comfort 15.1.0.0"; PictureOff "Navigates to SIMATIC PLC system diagnostics for TP700 Comfort 15.1.0.0"
   Button "HmiScreenItemData_1" at 23,190 size 159x47; TextOn 'Project information'; TextOff 'Project information'; PictureOn "Navigates to Project information for TP700 Comfort 15.1.0.0"; PictureOff "Navigates to Project information for TP700 Comfort 15.1.0.0"
   Button "HmiScreenItemData_2" at 23,249 size 159x47; TextOn 'System settings'; TextOff 'System settings'; PictureOn "Navigates to System settings for TP700 Comfort 15.1.0.0"; PictureOff "Navigates to System settings for TP700 Comfort 15.1.0.0"
   Button "HmiScreenItemData_3" at 23,308 size 159x47; TextOn 'User administration'; TextOff 'User administration'; PictureOn "Navigates to User administration for TP700 Comfort 15.1.0.0"; PictureOff "Navigates to User administration for TP700 Comfort 15.1.0.0"
      on Release: ActivateScreen("User administration", 0)
   Button "HmiScreenItemData_4" at 194,131 size 159x47; TextOn 'System information'; TextOff 'System information'; PictureOn "Navigates to System information for TP700 Comfort 15.1.0.0"; PictureOff "Navigates to System information for TP700 Comfort 15.1.0.0"
   Button "HmiScreenItemData_5" at 194,190 size 159x47; TextOn 'Different jobs'; TextOff 'Different jobs'; PictureOn "Navigates to Different jobs for TP700 Comfort 15.1.0.0"; PictureOff "Navigates to Different jobs for TP700 Comfort 15.1.0.0"
   Button "Calibrate screen" at 609,249 size 159x47; TextOn 'Calibrate screen'; TextOff 'Calibrate screen'
      on Release: function_bc3e350c()
   Button "Clean screen" at 609,308 size 159x47; TextOn 'Clean screen'; TextOff 'Clean screen'
      on Release: function_be740847(30)
   Button "Online" at 438,131 size 159x47; TextOn 'Online'; TextOff 'Online'
      on Release: function_bb44b551(0)
   Button "Offline" at 438,190 size 159x47; TextOn 'Offline'; TextOff 'Offline'
      on Release: function_bb44b551(1)
   Button "Transfer" at 438,249 size 159x47; TextOn 'Transfer'; TextOff 'Transfer'
      on Release: function_bb44b551(2)
   Button "Toggle language" at 438,308 size 159x47; TextOn 'Toggle language'; TextOff 'Toggle language'
      on Release: function_fb9197e8(-1)
   Button "Control Panel" at 609,131 size 159x47; TextOn 'Control Panel'; TextOff 'Control Panel'
      on Release: function_f34a74f3()
   Button "Stop Runtime" at 609,190 size 159x47; TextOn 'Stop Runtime'; TextOff 'Stop Runtime'
      on Release: StopRuntime(0)
   Button "Button_10" at 6,52 size 739x52; TextOff 'Enable'
   Button "Button_13" at 747,52 size 50x52; TextOff 'CmValveCtrl'; PictureOff "Home"
      on Release: ActivateScreen("Main_Screen", 0)

screen "Main_Screen" 800x480
   Button "Button_1" at 34,147 size 150x90; TextOff 'CmDriveSerPos'
      on Release: ActivateScreen("Screen_1", 0)
   Button "Button_10" at 6,52 size 785x52; TextOff 'Enable'
   TextField "Text field_8" at 346,17 size 107x23; Text 'Mainscreen'
   Button "Button_2" at 452,147 size 150x90; TextOff 'CmCommon'
   Button "Button_3" at 452,257 size 150x90; TextOff 'HMI Settings'
      on Release: ActivateScreen("HMI_Settings", 0)
   DateTimeField "HmiScreenItemData" at 695,23 size 105x30
   DateTimeField "HmiScreenItemData_1" at 695,0 size 105x30
   Button "Button_4" at 212,244 size 150x90; TextOff 'Change Mode'
      on Release: ResetBit("DB_CmDrvSerPos_CD_Commands_ModeChange")
      on Press: SetBit("DB_CmDrvSerPos_CD_Commands_ModeChange")
   IOField "I/O field_1" at 260,387 size 62x58; FormatPattern 9
      ProcessValue <- "VIS_CmDrvSerPos_stc_SD_iModeActual"
   TextField "Text field_1" at 34,326 size 134x23; Text '0 = Undefined'
   TextField "Text field_2" at 34,349 size 138x23; Text '1 = AutoInline'
   TextField "Text field_3" at 34,373 size 187x23; Text '2 = AutoStandalone'
   TextField "Text field_4" at 34,396 size 107x23; Text '3 = Manual'
   TextField "Text field_5" at 34,419 size 108x23; Text '4 = Service'
   TextField "Text field_6" at 34,440 size 139x23; Text '5 = SingleStep'
   IOField "I/O field_2" at 133,259 size 62x58; FormatPattern 9
      ProcessValue <- "DB_CmDrvSerPos_CD_iModeSet"
   TextField "Text field_7" at 35,275 size 96x23; Text 'Set Mode:'
   TextField "Text field_9" at 234,361 size 124x23; Text 'Actual Mode:'
   Ellipse "Ellipse_7" at 197,176 size 28x28
      Appearance <- "di_FeedbackEmStop"
   TextField "Text field_10" at 232,179 size 143x23; Text 'EM-Stop Active'

screen "User administration" 800x480
   UserView "HmiScreenItemData" at 4,4 size 740x475
   Button "Button_13" at 747,52 size 50x52; TextOff 'CmValveCtrl'; PictureOff "Home"
      on Release: ActivateScreen("Main_Screen", 0)

screen "Screen_3" 800x480, template "Template_1"
   TextField "Text field_3" at 525,122 size 60x23; Text 'Limits'
   IOField "I/O field_1" at 577,165 size 141x39; FormatPattern s999.9; Unit mm
      ProcessValue <- "VIS_CmDrvSerPos_stc_Settings_rSpLimitH_Units"
   TextField "Text field_6" at 385,172 size 98x23; Text 'Sp Limit H'
   TextField "Text field_7" at 385,217 size 95x23; Text 'Sp Limit L'
   Button "Button_10" at 6,52 size 739x52; TextOff 'Enable'
   TextField "Text field_8" at 315,17 size 143x23; Text 'CmDriveSerPos'
   Button "Button_11" at 747,417 size 51x56; TextOff 'Enable'; PictureOff "Down_Arrow"
      on Release: ActivateScreen("Screen_1", 0)
   Button "Button_12" at 747,112 size 51x56; TextOff 'Enable'; PictureOff "Up_Arrow"
      on Release: ActivateScreen("Screen_2", 0)
   TextField "Text field_10" at 772,280 size 16x23; Text '3'
   TextField "Text field_11" at 751,280 size 16x23; Text '3'
   Button "Button_13" at 747,52 size 50x52; TextOff 'CmValveCtrl'; PictureOff "Home"
      on Release: ActivateScreen("Main_Screen", 0)
   IOField "I/O field_2" at 577,209 size 141x39; FormatPattern s999.9; Unit mm
      ProcessValue <- "VIS_CmDrvSerPos_stc_Settings_rSpLimitL_Units"
   IOField "I/O field_4" at 578,253 size 141x39; FormatPattern s999.9; Unit mm
      ProcessValue <- "VIS_CmDrvSerPos_stc_Settings_rSpPositionOffset_Units"
   TextField "Text field_5" at 386,260 size 167x23; Text 'Calibration Offset'
   TextField "Text field_13" at 386,305 size 89x23; Text 'Unit type'
   IOField "I/O field_5" at 578,297 size 141x39; FormatPattern 9
      ProcessValue <- "VIS_CmDrvSerPos_stc_Settings_iSetUnits"
*)